PROGRAM main
  VAR
    HS101A_Open AT %IX0.0 : BOOL; (* Door open command pushbutton (NO) *)
    HS101B_Close AT %IX0.1 : BOOL; (* Door close command pushbutton (NO) *)
    ZSH101_Up AT %IX0.2 : BOOL; (* Door full-open limit switch (NO) *)
    ZSL101_Down AT %IX0.3 : BOOL; (* Door full-closed limit switch (NO) *)
    M101A_FWD AT %QX0.0 : BOOL; (* Motor forward (raise) contactor *)
    M101B_REV AT %QX0.1 : BOOL; (* Motor reverse (lower) contactor *)
  END_VAR

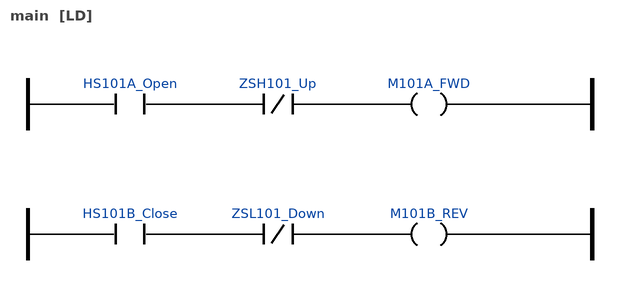
(* LD diagram, written out as Structured Text *)
M101A_FWD := HS101A_Open AND NOT ZSH101_Up;
M101B_REV := HS101B_Close AND NOT ZSL101_Down;
END_PROGRAM
